FUNCTION_BLOCK Basic1 (* Basic Function Block Type *)
  (* Standard: 61499-2 *)
  (* Version 0.0, 10/8/2026, Schneider Electric, Template *)
  PACKAGE Main;
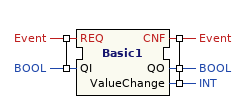
  EVENT_INPUT
    REQ WITH QI; (* Normal Execution Request *)
  END_EVENT
  EVENT_OUTPUT
    CNF WITH QO, ValueChange; (* Execution Confirmation *)
  END_EVENT
  VAR_INPUT
    QI : BOOL; (* Input event qualifier *)
  END_VAR
  VAR_OUTPUT
    QO : BOOL; (* Output event qualifier *)
    ValueChange : INT;
  END_VAR
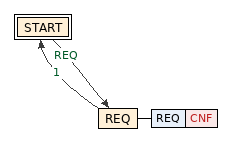
  EC_STATES
    START; (* Initial State *)
    REQ : REQ -> CNF;
  END_STATES
  EC_TRANSITIONS
    START TO REQ := REQ;
    REQ TO START := 1;
  END_TRANSITIONS
  ALGORITHM INIT IN ST: (* Initialization algorithm *)
;
  END_ALGORITHM
  ALGORITHM REQ IN ST: (* Normally executed algorithm *)
IF QO <> FALSE THEN
	ValueChange := 1;
END_IF;
;
  END_ALGORITHM
END_FUNCTION_BLOCK
